// TwinCAT 3 PLC project FB_BannerK50
// Title: FB_BannerK50
// Company: MBPersonalDev
// Author: mbragas
// ProjectVersion: 4.4.2025.01
// Description: Banner Engineering K50RGB IO Link
// ProgramVersion: 3.1.4023.0
// libraries:
//   Tc2_Standard, * (Beckhoff Automation GmbH)
//   Tc2_System, * (Beckhoff Automation GmbH)
//   Tc3_Module, * (Beckhoff Automation GmbH)
// project tree:
//   / PlcTask.TcTTO
//   POUs/FB_BannerK50/DUTs/ ST_Colors_Auto.TcDUT (not stored), ST_ProcessData_Manual.TcDUT (not stored), ST_ProcessValues.TcDUT
//   POUs/FB_BannerK50/ FB_BannerK50.TcPOU
//   POUs/ MAIN.TcPOU
//   Project Information/ F_GetCompany.TcPOU, F_GetTitle.TcPOU, F_GetVersion.TcPOU
//   Version/ Global_Version.TcGVL
// real-time tasks:
//   TASK PlcTask: cycle T#10ms, priority 20, ADS port 350
// I/O:
//   DEVICE Device 1 (EtherCAT), AmsNetId 192.168.1.165.2.1
//     Term 1 (EK1100) [EK1100 EtherCAT Coupler (2A E-Bus)]
//     Box 3 (ifm IO-Link Master AL1330) [ifm IO-Link Master AL1330]
//       modules: Module 1 (IOL_Out_4Byte), Module 2 (Deactivated), Module 3 (Deactivated), Module 4 (Deactivated)
//     Box 2 (EP1008-0001) [EP1008-0001 8 Ch. Dig. Input 24V, 3ms, M8]

CONFIGURATION FB_BannerK50
    RESOURCE PLC ON TwinCAT3
        TASK PlcTask(INTERVAL := T#10ms, PRIORITY := 20);
        PROGRAM MAIN WITH PlcTask : MAIN;
    END_RESOURCE
END_CONFIGURATION

// ---- POUs/FB_BannerK50/DUTs/ST_ProcessValues.TcDUT
TYPE ST_ProcessValues :
STRUCT
	//Byte 0 - Color 2 Intensity									// Binary Value
    High_Intensity					:	USINT	:= 0;				// 0000
    Medium_Intensity				:	USINT	:= 2;				// 0010
    Low_Intensity       			:	USINT	:= 1;				// 0001
    OFF_Intensity					:	USINT	:= 4;				// 0100
    
    //Byte 1 - Color 1 Animation & Intensity
    Steady_HighInt       			:	USINT	:= 1;				//	0001
    Flash_HighInt        			:	USINT	:= 2;				//	0010
    TwoFlash_HighInt        		:	USINT	:= 3;				//	0011
    Strobe_HighInt        			:	USINT	:= 4;				//	0100
    Half_HighInt        			:	USINT	:= 5;				//	0101
    HalfRotate_HighInt      		:	USINT	:= 6;				//	0110
    Chase_HighInt					:	USINT 	:= 7;				//	0111
    
    //Byte 2 - Rotation, Audible & Color 2
	AudibleOFF						:	USINT	:= 0;				//  0000
    AudibleSolid					: 	USINT	:= 32;				//	0010 0000
    AudiblePulse					: 	USINT	:= 64;				//	0100 0000
    
    //Byte 3 - Color & Flash Rate
    Green							:	USINT 	:= 0;				//  0
    Red								:	USINT 	:= 1;				//  0001	
    Orange							:	USINT 	:= 2;				//	0010
    Yellow							:	USINT 	:= 3;				//	0011
    Lime_Green						:	USINT 	:= 4;				//	0100
    Spring_Green					:	USINT 	:= 5;				//	0101
    Cyan							:	USINT 	:= 6;				//	0110
    SkyBlue							:	USINT 	:= 7;				//	0111
    Blue							:	USINT 	:= 8;				//	1111
    Violet							:	USINT 	:= 9;				//	1001
    Magenta							:	USINT 	:= 10;              //	1010
    Rose							:	USINT 	:= 11;              //	1011
    White							:	USINT 	:= 12;              //	1100
END_STRUCT
END_TYPE

// ---- Version/Global_Version.TcGVL
{attribute 'TcGenerated'}
{attribute 'no-analysis'}
{attribute 'linkalways'}
// This function has been automatically generated from the project information.
VAR_GLOBAL CONSTANT
	{attribute 'const_non_replaced'}
	stLibVersion_FB_BannerK50 : ST_LibVersion := (iMajor := 4, iMinor := 4, iBuild := 2025, iRevision := 1, nFlags := 0, sVersion := '4.4.2025.1');
END_VAR

// ---- POUs/MAIN.TcPOU
PROGRAM MAIN
VAR
	fbBanner			: FB_BannerK50;
END_VAR

fbBanner();

END_PROGRAM

// ---- POUs/FB_BannerK50/FB_BannerK50.TcPOU
FUNCTION_BLOCK FB_BannerK50
VAR_INPUT																									//		https://www.bannerengineering.com/us/en/products/part.802164.html  >>>>------ IO Link Data Reference Guide >>> Found Here
	AutoMode						:	BOOL := FALSE;
	SetAllFalse						:	BOOL := FALSE;
	
	// Structures
	Color							:	ST_Colors_Auto;
	Data							:	ST_ProcessData_Manual;
	Value							:   ST_ProcessValues;	
END_VAR

VAR_OUTPUT
	// IO
	Banner_Indicator 		AT %Q*  : 	ARRAY[0..3] OF USINT;
END_VAR

VAR
	ManualMode						:	BOOL := FALSE;				// To use Manual Mode, just call the FB
END_VAR

(*

Subindex 			     Name						Number of Bits 											Data Values


------------|------------------------------------|----------------|--------------------------------------------------------------------------------------------------------------------------------------
			|                        			 |                |
			|                        			 |                |
		1 	|		Color 1  					 |		5 		  |			0 = Green, 1 = Red, 2 = Orange, 3 = Yellow, 4 = Lime Green, 5 = Spring Green, 6 = Cyan, 7 = Sky Blue,
			|			 						 |	 	  		  |			8 = Blue, 9 = Violet, 10 = Magenta, 11 = Rose, 12 = White, 13 = Custom1, 14 = Custom2, 15 = Custom3,
			|			 						 |	  	  		  |			16 = Custom4, 17 = Custom5
						 						 |                |
------------|------------------------------------|----------------|--------------------------------------------------------------------------------------------------------------------------------------
			|                                    |                |
		2	|		Color Flash Rate (Hz)		 |		3 		  |			0 = 1.5, 1 = 0.5, 2 = 3.0, 3 = 6.0, 4 = 9.0, 5 = 12.0, 6=Custom
			|                                    |                |
------------|------------------------------------|----------------|--------------------------------------------------------------------------------------------------------------------------------------
			|                        			 |                |
		3	|		Color	 					 |	5	  		  |			0 = Green, 1 = Red, 2 = Orange, 3 = Yellow, 4 = Lime Green, 5 = Spring Green, 6 = Cyan, 7 = Sky Blue,
			|	                 				 |                |         8 = Blue, 9 = Violet, 10 = Magenta, 11 = Rose, 12 = White, 13 = Custom1, 14 = Custom2, 15 = Custom3,
		 	|			 						 |                |         16 = Custom4, 17 = Custom5
			|									 |		  		  |	
------------|------------------------------------|----------------|--------------------------------------------------------------------------------------------------------------------------------------
			|									 |				  |	
		4	|		Audible Mode (K50L2 Only)	 |		2 		  |			0 = Off, 1 = On, 2 = Pulse
		 	|                                    |                |
------------|------------------------------------|----------------|--------------------------------------------------------------------------------------------------------------------------------------
			|                                    |                |
		5	|		Rotation Direction		     |		1		  |			0 = CCW, 1 = CW
		    |                                    |                |
------------|------------------------------------|----------------|--------------------------------------------------------------------------------------------------------------------------------------
			|                                    |                |
		6	|		Animation Type				 |		4		  |			0 = Off, 1 = Steady, 2 = Flash, 3 = Two Flash, 4 = Strobe, 5 = Half/Half, 6 = Half/Half Rotate, 7 = Chase, 8 = Demo Mode
			|                                    |                |
------------|------------------------------------|----------------|--------------------------------------------------------------------------------------------------------------------------------------
			|                                    |                |
		7	|		Color 1 Intensity			 |		4		  |			0 = High, 1 = Low, 2 = Medium, 3 = Custom, 4 = Off
			|                                    |                |
------------|------------------------------------|----------------|--------------------------------------------------------------------------------------------------------------------------------------
		    |                                    |                |
		8  	|		Color 2 Intensity			 |		4 		  |			0 = High, 1 = Low, 2 = Medium, 3 = Custom, 4 = Off
		    |                                    |                |
------------|------------------------------------|----------------|--------------------------------------------------------------------------------------------------------------------------------------

*)

IF AutoMode THEN
	_M_SetColorAuto();
	ManualMode := FALSE;
ELSE
	_M_SetColorManual();
	ManualMode := TRUE;
	AutoMode   := FALSE;
END_IF

IF SetAllFalse THEN
	_M_SetAllFalse();
	SetAllFalse := FALSE;
END_IF

METHOD PRIVATE _M_SetAllFalse : BOOL
VAR_INPUT
END_VAR
//Green
Color.Green_Solid							:= FALSE;
Color.GreenSolid_AudibleSolid				:= FALSE;
Color.GreenSolid_AudiblePulse				:= FALSE;
Color.Green_Flash							:= FALSE;
Color.GreenFlash_AudibleSolid				:= FALSE;
Color.GreenFlash_AudiblePulse				:= FALSE;
                                	
//Red                           	
Color.Red_Solid								:= FALSE;
Color.RedSolid_AudibleSolid					:= FALSE;
Color.RedSolid_AudiblePulse					:= FALSE;
Color.Red_Flash								:= FALSE;
Color.RedFlash_AudibleSolid					:= FALSE;
Color.RedFlash_AudiblePulse					:= FALSE;
                                	
//Orange                        	
Color.Orange_Solid							:= FALSE;
Color.OrangeSolid_AudibleSolid				:= FALSE;
Color.OrangeSolid_AudiblePulse				:= FALSE;
Color.Orange_Flash							:= FALSE;
Color.OrangeFlash_AudibleSolid				:= FALSE;
Color.OrangeFlash_AudiblePulse				:= FALSE;
                                	
//Yellow                        	
Color.Yellow_Solid							:= FALSE;
Color.YellowSolid_AudibleSolid				:= FALSE;
Color.YellowSolid_AudiblePulse				:= FALSE;
Color.Yellow_Flash							:= FALSE;
Color.YellowFlash_AudibleSolid				:= FALSE;
Color.YellowFlash_AudiblePulse				:= FALSE;
                                	
//Lime Green                    	
Color.LimeGreen_Solid						:= FALSE;
Color.LimeGreenSolid_AudibleSolid			:= FALSE;
Color.LimeGreenSolid_AudiblePulse			:= FALSE;
Color.LimeGreen_Flash						:= FALSE;
Color.LimeGreenFlash_AudibleSolid			:= FALSE;
Color.LimeGreenFlash_AudiblePulse			:= FALSE;
                                	
//Spring Green                  	
Color.SpringGreen_Solid						:= FALSE;
Color.SpringGreenSolid_AudibleSolid			:= FALSE;
Color.SpringGreenSolid_AudiblePulse			:= FALSE;
Color.SpringGreen_Flash						:= FALSE;
Color.SpringGreenFlash_AudibleSolid			:= FALSE;
Color.SpringGreenFlash_AudiblePulse			:= FALSE;
                                	
//Cyan                          	
Color.Cyan_Solid							:= FALSE;
Color.CyanSolid_AudibleSolid				:= FALSE;
Color.CyanSolid_AudiblePulse				:= FALSE;
Color.Cyan_Flash							:= FALSE;
Color.CyanFlash_AudibleSolid				:= FALSE;
Color.CyanFlash_AudiblePulse				:= FALSE;
                                	
//Sky Blue                      	
Color.SkyBlue_Solid							:= FALSE;
Color.SkyBlueSolid_AudibleSolid				:= FALSE;
Color.SkyBlueSolid_AudiblePulse				:= FALSE;
Color.SkyBlue_Flash							:= FALSE;
Color.SkyBlueFlash_AudibleSolid				:= FALSE;
Color.SkyBlueFlash_AudiblePulse				:= FALSE;
                                	
//Blue                          	
Color.Blue_Solid							:= FALSE;
Color.BlueSolid_AudibleSolid				:= FALSE;
Color.BlueSolid_AudiblePulse				:= FALSE;
Color.Blue_Flash							:= FALSE;
Color.BlueFlash_AudibleSolid				:= FALSE;
Color.BlueFlash_AudiblePulse				:= FALSE;
                                	
//Violet                        	
Color.Violet_Solid							:= FALSE;
Color.VioletSolid_AudibleSolid				:= FALSE;
Color.VioletSolid_AudiblePulse				:= FALSE;
Color.Violet_Flash							:= FALSE;
Color.VioletFlash_AudibleSolid				:= FALSE;
Color.VioletFlash_AudiblePulse				:= FALSE;
                                	
//Magenta                       	
Color.Magenta_Solid							:= FALSE;
Color.MagentaSolid_AudibleSolid				:= FALSE;
Color.MagentaSolid_AudiblePulse				:= FALSE;
Color.Magenta_Flash							:= FALSE;
Color.MagentaFlash_AudibleSolid				:= FALSE;
Color.MagentaFlash_AudiblePulse				:= FALSE;
                                	
//Rose                          	
Color.Rose_Solid							:= FALSE;
Color.RoseSolid_AudibleSolid				:= FALSE;
Color.RoseSolid_AudiblePulse				:= FALSE;
Color.Rose_Flash							:= FALSE;
Color.RoseFlash_AudibleSolid				:= FALSE;
Color.RoseFlash_AudiblePulse				:= FALSE;
                                	
//White                         	
Color.WhiteFlash_AudiblePulse				:= FALSE;
                                	
//Demo Mode                     	
Color.Demo									:= FALSE;
                                	
//OFF                           	
Color.OFF									:= FALSE;
END_METHOD

METHOD PRIVATE _M_SetColorAuto : BOOL
VAR_INPUT
END_VAR
IF Automode AND NOT ManualMode THEN	
	IF Color.Green_Solid THEN
			Banner_Indicator[0] := 0;
			Banner_Indicator[1] := 1;
			Banner_Indicator[2] := 0;
			Banner_Indicator[3] := 0;
		
		ELSIF Color.GreenSolid_AudibleSolid THEN
			Banner_Indicator[0] := 0;
		    Banner_Indicator[1] := 1;
		    Banner_Indicator[2] := 32;
		    Banner_Indicator[3] := 0;
			
		ELSIF Color.GreenSolid_AudiblePulse THEN	
			Banner_Indicator[0] := 0;	
		   	Banner_Indicator[1] := 1;	
		   	Banner_Indicator[2] := 64;	
		   	Banner_Indicator[3] := 0;	
			
		ELSIF Color.Green_Flash THEN
			Banner_Indicator[0] := 0;
		    Banner_Indicator[1] := 2;
		    Banner_Indicator[2] := 0;
		    Banner_Indicator[3] := 0;
			
		ELSIF Color.GreenFlash_AudibleSolid THEN
			Banner_Indicator[0] := 0;
		    Banner_Indicator[1] := 2;
		    Banner_Indicator[2] := 32;
		    Banner_Indicator[3] := 0;
			
		ELSIF Color.GreenFlash_AudiblePulse THEN	
			Banner_Indicator[0] := 0;	
		    Banner_Indicator[1] := 2;	
		    Banner_Indicator[2] := 64;	
		    Banner_Indicator[3] := 0;	
			
		//Red Variations ---------------------------------------------------------------
		
		ELSIF Color.Red_Solid THEN
			Banner_Indicator[0] := 0;
			Banner_Indicator[1] := 1;
			Banner_Indicator[2] := 0;
			Banner_Indicator[3] := 1;
		
		ELSIF Color.RedSolid_AudibleSolid THEN
			Banner_Indicator[0] := 0;
		    Banner_Indicator[1] := 1;
		    Banner_Indicator[2] := 32;
		    Banner_Indicator[3] := 1;
		
		ELSIF Color.RedSolid_AudiblePulse THEN	
			Banner_Indicator[0] := 0;	
		    Banner_Indicator[1] := 1;	
		    Banner_Indicator[2] := 64;	
		    Banner_Indicator[3] := 1;	
			
		ELSIF Color.Red_Flash THEN
			Banner_Indicator[0] := 0;
		    Banner_Indicator[1] := 2;
		    Banner_Indicator[2] := 0;
		    Banner_Indicator[3] := 1;
	
		ELSIF Color.RedFlash_AudibleSolid THEN
			Banner_Indicator[0] := 0;
		    Banner_Indicator[1] := 2;
		    Banner_Indicator[2] := 32;
		    Banner_Indicator[3] := 1;
		
		ELSIF Color.RedFlash_AudiblePulse THEN	
			Banner_Indicator[0] := 0;	
		    Banner_Indicator[1] := 2;	
		    Banner_Indicator[2] := 64;	
		    Banner_Indicator[3] := 1;	
			
		//Orange Variations -------------------------------------------------------------	
			
		ELSIF Color.Orange_Solid THEN
			Banner_Indicator[0] := 0;
			Banner_Indicator[1] := 1;
			Banner_Indicator[2] := 0;
			Banner_Indicator[3] := 2;
		
		ELSIF Color.OrangeSolid_AudibleSolid THEN	
			Banner_Indicator[0] := 0;
		    Banner_Indicator[1] := 1;
		    Banner_Indicator[2] := 32;
		    Banner_Indicator[3] := 2;
		
		ELSIF Color.OrangeSolid_AudiblePulse THEN
			Banner_Indicator[0] := 0;	
		    Banner_Indicator[1] := 1;	
		    Banner_Indicator[2] := 64;	
		    Banner_Indicator[3] := 2;	
			
		ELSIF Color.Orange_Flash THEN	
			Banner_Indicator[0] := 0;
		    Banner_Indicator[1] := 2;
		    Banner_Indicator[2] := 0;
		    Banner_Indicator[3] := 2;
		
		ELSIF Color.OrangeFlash_AudibleSolid THEN
			Banner_Indicator[0] := 0;
		    Banner_Indicator[1] := 2;
		    Banner_Indicator[2] := 32;
		    Banner_Indicator[3] := 2;
			
		ELSIF Color.OrangeFlash_AudiblePulse THEN
			Banner_Indicator[0] := 0;	
		    Banner_Indicator[1] := 2;	
		    Banner_Indicator[2] := 64;	
		    Banner_Indicator[3] := 2;	

		//Yellow Variations -------------------------------------------------------------
		
		ELSIF Color.Yellow_Solid THEN            
			Banner_Indicator[0] := 0;               
			Banner_Indicator[1] := 1;               
			Banner_Indicator[2] := 0;               
			Banner_Indicator[3] := 3;               
	                                             
		ELSIF Color.YellowSolid_AudibleSolid THEN
			Banner_Indicator[0] := 0;               
		    Banner_Indicator[1] := 1;            
		    Banner_Indicator[2] := 32;            
		    Banner_Indicator[3] := 3;            
		                                         
		ELSIF Color.YellowSolid_AudiblePulse THEN
			Banner_Indicator[0] := 0;	              
		    Banner_Indicator[1] := 1;	           
		    Banner_Indicator[2] := 64;	           
		    Banner_Indicator[3] := 3;	           
			                                        
		ELSIF Color.Yellow_Flash THEN	           
			Banner_Indicator[0] := 0;               
		    Banner_Indicator[1] := 2;            
		    Banner_Indicator[2] := 0;            
		    Banner_Indicator[3] := 3;            
		                                         
		ELSIF Color.YellowFlash_AudibleSolid THEN
			Banner_Indicator[0] := 0;               
		    Banner_Indicator[1] := 2;            
		    Banner_Indicator[2] := 32;            
		    Banner_Indicator[3] := 3;            
			                                        
		ELSIF Color.YellowFlash_AudiblePulse THEN
			Banner_Indicator[0] := 0;	              
		    Banner_Indicator[1] := 2;	           
		    Banner_Indicator[2] := 64;	           
		    Banner_Indicator[3] := 3;	           

		//Lime Green Variations -------------------------------------------------------------
			
		ELSIF Color.LimeGreen_Solid THEN            	
			Banner_Indicator[0] := 0;               	
			Banner_Indicator[1] := 1;               	
			Banner_Indicator[2] := 0;               	
			Banner_Indicator[3] := 4;               	
		                                         	
		ELSIF Color.LimeGreenSolid_AudibleSolid THEN	
			Banner_Indicator[0] := 0;               	
		    Banner_Indicator[1] := 1;            	
		    Banner_Indicator[2] := 32;            	
		    Banner_Indicator[3] := 4;            	
		                                         	
		ELSIF Color.LimeGreenSolid_AudiblePulse THEN	
			Banner_Indicator[0] := 0;	              	
		    Banner_Indicator[1] := 1;	           	
		    Banner_Indicator[2] := 64;	           	
		    Banner_Indicator[3] := 4;	           	
			                                        	
		ELSIF Color.LimeGreen_Flash THEN	           	
			Banner_Indicator[0] := 0;               	
		    Banner_Indicator[1] := 2;            	
		    Banner_Indicator[2] := 0;            	
		    Banner_Indicator[3] := 4;            	
		                                         	
		ELSIF Color.LimeGreenFlash_AudibleSolid THEN	
			Banner_Indicator[0] := 0;               	
		    Banner_Indicator[1] := 2;            	
		    Banner_Indicator[2] := 32;            	
		    Banner_Indicator[3] := 4;            	
			                                        	
		ELSIF Color.LimeGreenFlash_AudiblePulse THEN	
			Banner_Indicator[0] := 0;	              	
		    Banner_Indicator[1] := 2;	           	
		    Banner_Indicator[2] := 64;	           	
		    Banner_Indicator[3] := 4;	           	
			
		//Spring Green Variations -------------------------------------------------------------	
			
		ELSIF Color.SpringGreen_Solid THEN            	
			Banner_Indicator[0] := 0;               	
			Banner_Indicator[1] := 1;               	
			Banner_Indicator[2] := 0;               	
			Banner_Indicator[3] := 5;               	
		                                         	
		ELSIF Color.SpringGreenSolid_AudibleSolid THEN	
			Banner_Indicator[0] := 0;               	
		    Banner_Indicator[1] := 1;            	
		    Banner_Indicator[2] := 32;            	
		    Banner_Indicator[3] := 5;            	
		                                         	
		ELSIF Color.SpringGreenSolid_AudiblePulse THEN	
			Banner_Indicator[0] := 0;	              	
		    Banner_Indicator[1] := 1;	           	
		    Banner_Indicator[2] := 64;	           	
		    Banner_Indicator[3] := 5;	           	
			                                        	
		ELSIF Color.SpringGreen_Flash THEN	           	
			Banner_Indicator[0] := 0;               	
		    Banner_Indicator[1] := 2;            	
		    Banner_Indicator[2] := 0;            	
		    Banner_Indicator[3] := 5;            	
		                                         	
		ELSIF Color.SpringGreenFlash_AudibleSolid THEN	
			Banner_Indicator[0] := 0;               	
		    Banner_Indicator[1] := 2;            	
		    Banner_Indicator[2] := 32;            	
		    Banner_Indicator[3] := 5;            	
			                                        	
		ELSIF Color.SpringGreenFlash_AudiblePulse THEN	
			Banner_Indicator[0] := 0;	              	
		    Banner_Indicator[1] := 2;	           	
		    Banner_Indicator[2] := 64;	           	
		    Banner_Indicator[3] := 5;	           	
			
		//Cyan Variations -------------------------------------------------------------
        
        ELSIF Color.Cyan_Solid THEN            
        	Banner_Indicator[0] := 0;               
        	Banner_Indicator[1] := 1;               
        	Banner_Indicator[2] := 0;               
        	Banner_Indicator[3] := 6;               
                                                 
        ELSIF Color.CyanSolid_AudibleSolid THEN
        	Banner_Indicator[0] := 0;               
            Banner_Indicator[1] := 1;            
            Banner_Indicator[2] := 32;            
            Banner_Indicator[3] := 6;            
                                                 
        ELSIF Color.CyanSolid_AudiblePulse THEN
        	Banner_Indicator[0] := 0;	              
            Banner_Indicator[1] := 1;	           
            Banner_Indicator[2] := 64;	           
            Banner_Indicator[3] := 6;	           
        	                                        
        ELSIF Color.Cyan_Flash THEN	           
        	Banner_Indicator[0] := 0;               
            Banner_Indicator[1] := 2;            
            Banner_Indicator[2] := 0;            
            Banner_Indicator[3] := 6;            
                                                 
        ELSIF Color.CyanFlash_AudibleSolid THEN
        	Banner_Indicator[0] := 0;               
            Banner_Indicator[1] := 2;            
            Banner_Indicator[2] := 32;            
            Banner_Indicator[3] := 6;            
        	                                        
        ELSIF Color.CyanFlash_AudiblePulse THEN
        	Banner_Indicator[0] := 0;	              
            Banner_Indicator[1] := 2;	           
            Banner_Indicator[2] := 64;	           
            Banner_Indicator[3] := 6;	           

		//Sky Blue Variations -------------------------------------------------------------
        
        ELSIF Color.SkyBlue_Solid THEN            
        	Banner_Indicator[0] := 0;               
        	Banner_Indicator[1] := 1;               
        	Banner_Indicator[2] := 0;               
        	Banner_Indicator[3] := 7;               
                                                 
        ELSIF Color.SkyBlueSolid_AudibleSolid THEN
        	Banner_Indicator[0] := 0;               
            Banner_Indicator[1] := 1;            
            Banner_Indicator[2] := 32;            
            Banner_Indicator[3] := 7;            
                                                 
        ELSIF Color.SkyBlueSolid_AudiblePulse THEN
        	Banner_Indicator[0] := 0;	              
            Banner_Indicator[1] := 1;	           
            Banner_Indicator[2] := 64;	           
            Banner_Indicator[3] := 7;	           
        	                                        
        ELSIF Color.SkyBlue_Flash THEN	           
        	Banner_Indicator[0] := 0;               
            Banner_Indicator[1] := 2;            
            Banner_Indicator[2] := 0;            
            Banner_Indicator[3] := 7;            
                                                 
        ELSIF Color.SkyBlueFlash_AudibleSolid THEN
        	Banner_Indicator[0] := 0;               
            Banner_Indicator[1] := 2;            
            Banner_Indicator[2] := 32;            
            Banner_Indicator[3] := 7;            
        	                                        
        ELSIF Color.SkyBlueFlash_AudiblePulse THEN
        	Banner_Indicator[0] := 0;	              
            Banner_Indicator[1] := 2;	           
            Banner_Indicator[2] := 64;	           
            Banner_Indicator[3] := 7;	           

		//Blue Variations -------------------------------------------------------------
        
        ELSIF Color.Blue_Solid THEN            
        	Banner_Indicator[0] := 0;               
        	Banner_Indicator[1] := 1;               
        	Banner_Indicator[2] := 0;               
        	Banner_Indicator[3] := 8;               
                                                 
        ELSIF Color.BlueSolid_AudibleSolid THEN
        	Banner_Indicator[0] := 0;               
            Banner_Indicator[1] := 1;            
            Banner_Indicator[2] := 32;            
            Banner_Indicator[3] := 8;            
                                                 
        ELSIF Color.BlueSolid_AudiblePulse THEN
        	Banner_Indicator[0] := 0;	              
            Banner_Indicator[1] := 1;	           
            Banner_Indicator[2] := 64;	           
            Banner_Indicator[3] := 8;	           
        	                                        
        ELSIF Color.Blue_Flash THEN	           
        	Banner_Indicator[0] := 0;               
            Banner_Indicator[1] := 2;            
            Banner_Indicator[2] := 0;            
            Banner_Indicator[3] := 8;            
                                                 
        ELSIF Color.BlueFlash_AudibleSolid THEN
        	Banner_Indicator[0] := 0;               
            Banner_Indicator[1] := 2;            
            Banner_Indicator[2] := 32;            
            Banner_Indicator[3] := 8;            
        	                                        
        ELSIF Color.BlueFlash_AudiblePulse THEN
        	Banner_Indicator[0] := 0;	              
            Banner_Indicator[1] := 2;	           
            Banner_Indicator[2] := 64;	           
            Banner_Indicator[3] := 8;	           

		//Violet Variations -------------------------------------------------------------
        
        ELSIF Color.Violet_Solid THEN            
        	Banner_Indicator[0] := 0;               
        	Banner_Indicator[1] := 1;               
        	Banner_Indicator[2] := 0;               
        	Banner_Indicator[3] := 9;               
                                                 
        ELSIF Color.VioletSolid_AudibleSolid THEN
        	Banner_Indicator[0] := 0;               
            Banner_Indicator[1] := 1;            
            Banner_Indicator[2] := 32;            
            Banner_Indicator[3] := 9;            
                                                 
        ELSIF Color.VioletSolid_AudiblePulse THEN
        	Banner_Indicator[0] := 0;	              
            Banner_Indicator[1] := 1;	           
            Banner_Indicator[2] := 64;	           
            Banner_Indicator[3] := 9;	           
        	                                        
        ELSIF Color.Violet_Flash THEN	           
        	Banner_Indicator[0] := 0;               
            Banner_Indicator[1] := 2;            
            Banner_Indicator[2] := 0;            
            Banner_Indicator[3] := 9;            
                                                 
        ELSIF Color.VioletFlash_AudibleSolid THEN
        	Banner_Indicator[0] := 0;               
            Banner_Indicator[1] := 2;            
            Banner_Indicator[2] := 32;            
            Banner_Indicator[3] := 9;            
        	                                        
        ELSIF Color.VioletFlash_AudiblePulse THEN
        	Banner_Indicator[0] := 0;	              
            Banner_Indicator[1] := 2;	           
            Banner_Indicator[2] := 64;	           
            Banner_Indicator[3] := 9;	           

		//Magenta Variations -------------------------------------------------------------
        
        ELSIF Color.Magenta_Solid THEN            
        	Banner_Indicator[0] := 0;               
        	Banner_Indicator[1] := 1;               
        	Banner_Indicator[2] := 0;               
        	Banner_Indicator[3] := 10;               
                                                 
        ELSIF Color.MagentaSolid_AudibleSolid THEN
        	Banner_Indicator[0] := 0;               
            Banner_Indicator[1] := 1;            
            Banner_Indicator[2] := 32;            
            Banner_Indicator[3] := 10;            
	                                             
		ELSIF Color.MagentaSolid_AudiblePulse THEN	
			Banner_Indicator[0] := 0;	              	
		    Banner_Indicator[1] := 1;	           	
		    Banner_Indicator[2] := 64;	           	
		    Banner_Indicator[3] := 10;	           	
			                                        	
		ELSIF Color.Magenta_Flash THEN	           	
			Banner_Indicator[0] := 0;               	
		    Banner_Indicator[1] := 2;            	
		    Banner_Indicator[2] := 0;            	
		    Banner_Indicator[3] := 10;            
                                                 
        ELSIF Color.MagentaFlash_AudibleSolid THEN
        	Banner_Indicator[0] := 0;               
            Banner_Indicator[1] := 2;            
            Banner_Indicator[2] := 32;            
            Banner_Indicator[3] := 10;            
        	                                        
        ELSIF Color.MagentaFlash_AudiblePulse THEN
        	Banner_Indicator[0] := 0;	              
            Banner_Indicator[1] := 2;	           
            Banner_Indicator[2] := 64;	           
            Banner_Indicator[3] := 10;	           

		//Rose Variations -------------------------------------------------------------
        
        ELSIF Color.Rose_Solid THEN            
        	Banner_Indicator[0] := 0;               
        	Banner_Indicator[1] := 1;               
        	Banner_Indicator[2] := 0;               
        	Banner_Indicator[3] := 11;               
                                                 
        ELSIF Color.RoseSolid_AudibleSolid THEN
        	Banner_Indicator[0] := 0;               
            Banner_Indicator[1] := 1;            
            Banner_Indicator[2] := 32;            
            Banner_Indicator[3] := 11;            
                                                 
        ELSIF Color.RoseSolid_AudiblePulse THEN
        	Banner_Indicator[0] := 0;	              
            Banner_Indicator[1] := 1;	           
            Banner_Indicator[2] := 64;	           
            Banner_Indicator[3] := 11;	           
        	                                        
        ELSIF Color.Rose_Flash THEN	           
        	Banner_Indicator[0] := 0;               
            Banner_Indicator[1] := 2;            
            Banner_Indicator[2] := 0;            
            Banner_Indicator[3] := 11;            
                                                 
        ELSIF Color.RoseFlash_AudibleSolid THEN
        	Banner_Indicator[0] := 0;               
            Banner_Indicator[1] := 2;            
            Banner_Indicator[2] := 32;            
            Banner_Indicator[3] := 11;            
        	                                        
        ELSIF Color.RoseFlash_AudiblePulse THEN
        	Banner_Indicator[0] := 0;	              
            Banner_Indicator[1] := 2;	           
            Banner_Indicator[2] := 64;	           
            Banner_Indicator[3] := 11;	           

		//White Variations -------------------------------------------------------------
        
        ELSIF Color.White_Solid THEN            
        	Banner_Indicator[0] := 0;               
        	Banner_Indicator[1] := 1;               
        	Banner_Indicator[2] := 0;               
        	Banner_Indicator[3] := 12;               
                                                 
        ELSIF Color.WhiteSolid_AudibleSolid THEN
        	Banner_Indicator[0] := 0;               
            Banner_Indicator[1] := 1;            
            Banner_Indicator[2] := 32;            
            Banner_Indicator[3] := 12;            
                                                 
        ELSIF Color.WhiteSolid_AudiblePulse THEN
        	Banner_Indicator[0] := 0;	              
            Banner_Indicator[1] := 1;	           
            Banner_Indicator[2] := 64;	           
            Banner_Indicator[3] := 12;	           
        	                                        
        ELSIF Color.White_Flash THEN	           
        	Banner_Indicator[0] := 0;               
            Banner_Indicator[1] := 2;            
            Banner_Indicator[2] := 0;            
            Banner_Indicator[3] := 12;            
                                                 
        ELSIF Color.WhiteFlash_AudibleSolid THEN
        	Banner_Indicator[0] := 0;               
            Banner_Indicator[1] := 2;            
            Banner_Indicator[2] := 32;            
            Banner_Indicator[3] := 12;            
        	                                        
        ELSIF Color.WhiteFlash_AudiblePulse THEN
        	Banner_Indicator[0] := 0;	              
            Banner_Indicator[1] := 2;	           
            Banner_Indicator[2] := 64;	           
            Banner_Indicator[3] := 12;	           

		//Demo Variations -------------------------------------------------------------
        
        ELSIF Color.Demo THEN            
        	Banner_Indicator[0] := 0;               
        	Banner_Indicator[1] := 8;               
        	Banner_Indicator[2] := 0;               
        	Banner_Indicator[3] := 0;               
        
		//OFF
                                         
		ELSIF Color.OFF THEN           
			Banner_Indicator[0] := 0;   	
			Banner_Indicator[1] := 0;   	
			Banner_Indicator[2] := 0;   	
			Banner_Indicator[3] := 0;   	
	ELSE
		Banner_Indicator[0] := 0;
        Banner_Indicator[1] := 0;
        Banner_Indicator[2] := 0;
        Banner_Indicator[3] := 0;
		_M_SetAllFalse();
	END_IF
END_IF
END_METHOD

METHOD PRIVATE _M_SetColorManual : BOOL
VAR_INPUT
END_VAR
IF ManualMode AND NOT AutoMode THEN
	 Banner_Indicator[0]:= Data.Octet_0;
	 Banner_Indicator[1]:= Data.Octet_1;
	 Banner_Indicator[2]:= Data.Octet_2;
	 Banner_Indicator[3]:= Data.Octet_3;
END_IF
END_METHOD

{reion "Property"}
PROPERTY P_Auto : REFERENCE TO ST_Colors_Auto;
GET
P_Auto REF= Color ;
END_GET
END_PROPERTY

PROPERTY P_Manual : REFERENCE TO ST_ProcessData_Manual;
GET
P_Manual REF= Data;
END_GET
END_PROPERTY

PROPERTY P_Values : REFERENCE TO ST_ProcessValues;
GET
P_Values REF= Value;
END_GET
END_PROPERTY

END_FUNCTION_BLOCK

// ---- Project Information/F_GetCompany.TcPOU
// This function has been automatically generated from the project information.
{attribute 'signature_flag' := '1073741824'}
{attribute 'TcGenerated'}
{attribute 'no-analysis'}
FUNCTION F_GetCompany : WSTRING
VAR_INPUT
	
END_VAR

F_GetCompany := "MBPersonalDev";

END_FUNCTION

// ---- Project Information/F_GetTitle.TcPOU
// This function has been automatically generated from the project information.
{attribute 'signature_flag' := '1073741824'}
{attribute 'TcGenerated'}
{attribute 'no-analysis'}
FUNCTION F_GetTitle : WSTRING
VAR_INPUT
	
END_VAR

F_GetTitle := "FB_BannerK50";

END_FUNCTION

// ---- Project Information/F_GetVersion.TcPOU
// This function has been automatically generated from the project information.
{attribute 'signature_flag' := '1073741824'}
{attribute 'TcGenerated'}
{attribute 'no-analysis'}
FUNCTION F_GetVersion : ST_LibVersion
VAR_INPUT
	
END_VAR

F_GetVersion.iMajor := 4;
F_GetVersion.iMinor := 4;
F_GetVersion.iBuild := 2025;
F_GetVersion.iRevision := 1;
F_GetVersion.sVersion := '4.4.2025.1';
F_GetVersion.nFlags := 0;

END_FUNCTION
